// TIA Portal V16 export
// export: Created 2024-09-05T17:39:13.1604731Z, ExportSetting WithDefaults, DisplayName Totally Integrated Automation Portal, DisplayVersion V16 Update 6, DisplayName TIA Portal Version Control Interface, DisplayVersion V16 Update 2, DisplayName TIA Portal Openness, DisplayVersion V16 Update 6, DisplayName STEP 7 Professional, DisplayVersion V16 Update 6, DisplayName STEP 7 Safety, DisplayVersion V16, DisplayName WinCC Advanced, DisplayVersion V16 Update 6
FUNCTION_BLOCK "Readings"   // FB300, LAD
{ S7_Optimized_Access := 'TRUE' }
VERSION : 0.1
// stored: AutoNumber false, IsIECCheckEnabled false, IsRetainMemResEnabled false, MemoryReserve 100, SetENOAutomatically false, UDAEnableTagReadback false
   VAR
      Stat : Struct
         Init : Bool;
         Run : Bool;
         Process : Bool;
      END_STRUCT;
   END_VAR
   VAR_TEMP
      i : Int;
   END_VAR
BEGIN

REGION Network 2 (SCL)
   FOR #i := 1 TO "MaxReader" DO
       IF "DB_ProductionProgramActual".Program.Readings[#i].Enable THEN
           IF "DB_ProductionProgramActual".Program.Readings[#i].ReaderNumber > 0 THEN
               "Reader Cognex Dataman"("Reader Parameters".Reader["DB_ProductionProgramActual".Program.Readings[#i].ReaderNumber]);



               ;
           END_IF;


       END_IF;

       ;
   END_FOR;
END_REGION
END_FUNCTION_BLOCK
